Staubli VAL3: RefreshList.pgx

program RefreshList()
  local num l_ni
begin
  //
  if bListRefresh
    sParameter[0]="j1"
    sParameter[1]="j2"
    sParameter[2]="j3"
    sParameter[3]="j4"
    sParameter[4]="j5"
    sParameter[5]="j6"
    //
    sListItemValue[0]=toString(".3",PublicData:jHome.j1)
    sListItemValue[1]=toString(".3",PublicData:jHome.j2)
    sListItemValue[2]=toString(".3",PublicData:jHome.j3)
    sListItemValue[3]=toString(".3",PublicData:jHome.j4)
    sListItemValue[4]=toString(".3",PublicData:jHome.j5)
    sListItemValue[5]=toString(".3",PublicData:jHome.j6)
  endIf

end
